PROGRAM LogicalCircuits_Ex10
VAR
	S1 					: DigitalInput_NO;
	S2 					: DigitalInput_NC;
	P1 					: DigitalOutput;
END_VAR

IF S1.isOn THEN
	P1.On();
END_IF
IF S2.broken THEN
	P1.Off();
END_IF

END_PROGRAM

(* stored: Version 1.1.0.1
   POU LogicalCircuits_Ex10: Id {47befc8f-72fb-4a91-825d-5f6b8795ce00}, SpecialFunc None *)
